{attribute 'enable_dynamic_creation'}
FUNCTION_BLOCK FutureMCReset EXTENDS FB_AbstructFuture
VAR_INPUT
END_VAR
VAR_OUTPUT
END_VAR
VAR
	_axis: REFERENCE TO AXIS_REF;
	_mc_reset	: MC_Reset;
	_error_id :HRESULT;
	_exec_state : UDINT;
END_VAR

METHOD execute : BOOL // Return TRUE if finish.

CASE _exec_state OF
	0:
		_mc_reset(axis := _axis, Execute := FALSE);
		_mc_reset(Axis:= _axis, Execute := TRUE );
		_exec_state := 1;
	1:
		IF _mc_reset.Busy THEN
			_mc_reset(Axis:= _axis,Execute := FALSE);
		END_IF
END_CASE

_error_id := _mc_reset.ErrorID;
execute := _mc_reset.Done OR _mc_reset.Error;
END_METHOD

METHOD init : BOOL // Return TRUE if finish.
_exec_state := 0;
init := TRUE;
END_METHOD

PROPERTY nErrorID : HRESULT
GET
nErrorID := _error_id;
END_GET
SET
END_SET
END_PROPERTY

METHOD set_parameters : BOOL
VAR_INPUT
	axis : REFERENCE TO AXIS_REF;
END_VAR
_axis REF= axis;
END_METHOD

END_FUNCTION_BLOCK

(* stored: Version 1.1.0.1, ProductVersion 3.1.4026.13
   POU FutureMCReset: Id {ee805a4a-5dfe-4650-9a98-91a6767180f3}, SpecialFunc None
   Method execute: Id {92464e08-2363-42d1-8525-536370e535b6}
   Method init: Id {83fe482e-32ec-4cb8-8167-dc39efd52913}
   Property nErrorID: Id {a880be76-8bd0-48c4-a77e-d3d6f9cb688f}
   Get Get: Id {802abbee-6aaf-42e2-bb73-83c390bd9c0b}
   Set Set: Id {0a0bed34-02c2-4cee-9f6b-40295d9a6828}
   Method set_parameters: Id {20e83138-9b09-4010-ae06-16dcf275b143} *)
